INTERFACE I_Drive_AX5000

METHOD DriveReset : BOOL
VAR_INPUT
END_VAR
END_METHOD

PROPERTY REF_Axis : REFERENCE TO AXIS_REF
GET
END_GET
SET
END_SET
END_PROPERTY

PROPERTY SercosErrorID : UINT
GET
END_GET
END_PROPERTY

END_INTERFACE

(* stored: Version 1.1.0.1, ProductVersion 3.1.4024.12
   Itf I_Drive_AX5000: Id {7a144353-44d3-483e-b59e-67643558209a}
   Method DriveReset: Id {bd897b02-233d-46c1-9be0-cc26f0f86b28}
   Property REF_Axis: Id {33062a85-b564-4044-a444-1072040d6d4c}
   Get Get: Id {2e8d1bcf-6f47-4a24-80c0-6dd306c6527f}
   Set Set: Id {3c24ff3d-6146-43cf-a7da-c33ab64a338b}
   Property SercosErrorID: Id {fe32639d-486c-42a7-b035-c6ea67b0a239}
   Get Get: Id {e4600d9f-0e53-40d8-a927-6c366a777ed5} *)
